(* IEC 61131-3 sources: esbmc-plcplus-llb-artifact/corpora/datasets/PLC_Defuser_dev/Datasets/SWAT/malicious/timer/ladder_timer/smal_timer1_82, 1 file *)

(* ---- smal_timer1_82.st ---- *)
PROGRAM PLC2
  VAR_INPUT
    level : DINT;
  END_VAR
  VAR_OUTPUT
    request : BOOL;
  END_VAR
  VAR
    open_req : BOOL;
    close_req : BOOL;
    low_2 : DINT := 10;
    high_2 : DINT := 20;
    _TMP_LE10_ENO : BOOL;
    _TMP_LE10_OUT : BOOL;
    _TMP_GE11_ENO : BOOL;
    _TMP_GE11_OUT : BOOL;
  END_VAR

  _TMP_LE10_OUT := LE(EN := TRUE, IN1 := level, IN2 := low_2, ENO => _TMP_LE10_ENO);
  open_req := _TMP_LE10_OUT;
  _TMP_GE11_OUT := GE(EN := TRUE, IN1 := level, IN2 := high_2, ENO => _TMP_GE11_ENO);
  close_req := _TMP_GE11_OUT;
  request := NOT(close_req) AND (open_req OR request);
END_PROGRAM

FUNCTION_BLOCK check_pumps
  VAR_INPUT
    IN1 : DINT;
    IN2 : DINT;
  END_VAR
  VAR_OUTPUT
    OUT : BOOL;
  END_VAR
  VAR
    i : INT;
  END_VAR

  if IN1 < IN2 then
    OUT:=TRUE;
  end_if;
  if IN1 >= IN2 then
    OUT:= FALSE;
  end_if;

  i:=0;
  while i< 4 do
      OUT:=FALSE;
  end_while;
END_FUNCTION_BLOCK

PROGRAM PLC1
  VAR_INPUT
    level : DINT;
    request : DINT;
  END_VAR
  VAR_OUTPUT
    pumps : BOOL;
    pumps_state : BOOL;
    valve : BOOL;
    real_value : DINT;
  END_VAR
  VAR
    low : BOOL;
    high : BOOL;
  END_VAR

  VAR
    open_req : BOOL;
    close_req : BOOL;
    low_1 : DINT := 40;
    high_1 : DINT := 80;
    check_pumps0 : check_pumps;
    TON0 : TON;
    _TMP_SUB39_ENO : BOOL;
    _TMP_SUB39_OUT : DINT;
    _TMP_LE3_ENO : BOOL;
    _TMP_LE3_OUT : BOOL;
    _TMP_GE7_ENO : BOOL;
    _TMP_GE7_OUT : BOOL;
    _TMP_EQ23_ENO : BOOL;
    _TMP_EQ23_OUT : BOOL;
    _TMP_EQ24_ENO : BOOL;
    _TMP_EQ24_OUT : BOOL;
  END_VAR

  _TMP_SUB39_OUT := SUB(EN := TRUE, IN1 := level, IN2 := 5, ENO => _TMP_SUB39_ENO);
  IF _TMP_SUB39_ENO THEN
      real_value := _TMP_SUB39_OUT;
  END_IF;
  _TMP_LE3_OUT := LE(EN := TRUE, IN1 := real_value, IN2 := low_1, ENO => _TMP_LE3_ENO);
  low := _TMP_LE3_OUT;
  _TMP_GE7_OUT := GE(EN := TRUE, IN1 := real_value, IN2 := high_1, ENO => _TMP_GE7_ENO);
  high := _TMP_GE7_OUT;
  TON0(IN := TRUE, PT := T#1000ms);
  check_pumps0(EN := TON0.Q, IN1 := level, IN2 := high_1);
  IF check_pumps0.ENO THEN
      pumps_state := check_pumps0.OUT;
  END_IF;
  _TMP_EQ23_OUT := EQ(EN := TRUE, IN1 := request, IN2 := 1, ENO => _TMP_EQ23_ENO);
  open_req := _TMP_EQ23_OUT;
  _TMP_EQ24_OUT := EQ(EN := TRUE, IN1 := request, IN2 := 0, ENO => _TMP_EQ24_ENO);
  close_req := _TMP_EQ24_OUT;
  pumps := NOT(high) AND (low OR pumps);
  valve := NOT(close_req) AND (open_req AND NOT(low) OR valve);
END_PROGRAM

PROGRAM PLC3
  VAR_INPUT
    level : DINT;
  END_VAR
  VAR_OUTPUT
    pump : BOOL;
  END_VAR
  VAR
    low : BOOL;
    high : BOOL;
    low_3 : DINT := 0;
    high_3 : DINT := 10;
    _TMP_LE13_ENO : BOOL;
    _TMP_LE13_OUT : BOOL;
    _TMP_GE12_ENO : BOOL;
    _TMP_GE12_OUT : BOOL;
  END_VAR

  _TMP_LE13_OUT := LE(EN := TRUE, IN1 := level, IN2 := low_3, ENO => _TMP_LE13_ENO);
  low := _TMP_LE13_OUT;
  _TMP_GE12_OUT := GE(EN := TRUE, IN1 := level, IN2 := high_3, ENO => _TMP_GE12_ENO);
  high := _TMP_GE12_OUT;
  pump := NOT(low) AND (high OR pump);
END_PROGRAM

CONFIGURATION Config0

  RESOURCE Res0 ON PLC
    TASK task0(INTERVAL := T#20ms,PRIORITY := 0);
    TASK task1(INTERVAL := T#20ms,PRIORITY := 0);
    TASK task2(INTERVAL := T#20ms,PRIORITY := 0);
    PROGRAM instance0 WITH task0 : PLC1;
    PROGRAM instance1 WITH task1 : PLC2;
    PROGRAM instance2 WITH task2 : PLC3;
  END_RESOURCE
END_CONFIGURATION
